// TwinCAT 3 PLC project Main
// ProgramVersion: 3.1.4023.0
// libraries:
//   Tc2_Standard, * (Beckhoff Automation GmbH)
//   Tc2_System, * (Beckhoff Automation GmbH)
//   Tc3_Module, * (Beckhoff Automation GmbH)
// project tree:
//   DUTs/ Controller.TcDUT, ControllerCmd.TcDUT, E_TriggerModes.TcDUT, E_PlayerID.TcDUT, E_ConnectionType.TcDUT, E_LedOptions.TcDUT, E_PulseOptions.TcDUT, E_Brightness.TcDUT, Point.TcDUT
//   GVLs/ Global.TcGVL
//   / PlcTask.TcTTO
//   POUs/ MAIN.TcPOU
// real-time tasks:
//   TASK PlcTask: cycle T#10ms, priority 20, ADS port 350

CONFIGURATION Main
    RESOURCE PLC ON TwinCAT3
        TASK PlcTask(INTERVAL := T#10ms, PRIORITY := 20);
        PROGRAM MAIN WITH PlcTask : MAIN;
    END_RESOURCE
END_CONFIGURATION

// ---- DUTs/Controller.TcDUT
TYPE Controller :
STRUCT
	LeftJoystickX : INT;
	LeftJoystickY : INT;
	RightJoystickX : INT;
	RightJoystickY : INT;
	LeftTrigger : INT;
	RightTrigger : INT;
	LeftBumper : BOOL;
	RightBumper : BOOL;
	ButtonTriangle : BOOL;
	ButtonCircle : BOOL;
	ButtonSquare : BOOL;
	ButtonCross : BOOL;
	LeftThumb : BOOL;
	RightThumb : BOOL;
	Share : BOOL;
	Options : BOOL;
	Ps : BOOL;
	DPadUp : BOOL;
	DPadDown : BOOL;
	DPadLeft : BOOL;
	DPadRight : BOOL;
	TouchBtn : BOOL;
	TrackPadTouch0Active : BOOL;
	TrackPadTouch1Active : BOOL;
	TrackPadTouch0ID : INT;
	TrackPadTouch1ID : INT;
	TrackPadTouch0X : INT;
	TrackPadTouch0Y : INT;
	TrackPadTouch1X : INT;
	TrackPadTouch1Y : INT;
	GyroPitch : INT;
	GyroYaw : INT;
	GyroRoll : INT;
	AccX : INT;
	AccY : INT;
	AccZ : INT;
	MicBtn : BOOL;
END_STRUCT
END_TYPE

// ---- DUTs/ControllerCmd.TcDUT
TYPE ControllerCmd :
STRUCT
	
	LedRed : INT := 255;
	LedGreen : INT;
	LedBlue : INT;
	Player : E_PlayerID;
	LedOptions : E_LedOptions;
	PulseOptions : E_PulseOptions;
	Brightness : E_Brightness;
	LeftHaptic : INT;
	RightHaptic : INT;
	LeftTriggerMode : E_TriggerModes;
	LeftTriggerLevel1 : INT;
	LeftTriggerLevel2 : INT;
	LeftTriggerLevel3 : INT;
	LeftTriggerLevel4 : INT;
	LeftTriggerLevel5 : INT;
	LeftTriggerLevel6 : INT;
	LeftTriggerLevel7 : INT;
	RightTriggerMode : E_TriggerModes;
	RightTriggerLevel1 : INT;
	RightTriggerLevel2 : INT;
	RightTriggerLevel3 : INT;
	RightTriggerLevel4 : INT;
	RightTriggerLevel5 : INT;
	RightTriggerLevel6 : INT;
	RightTriggerLevel7 : INT;
	MicLed : BOOL;
	MicMute : BOOL;
	
END_STRUCT
END_TYPE

// ---- DUTs/E_TriggerModes.TcDUT
{attribute 'qualified_only'}
TYPE E_TriggerModes :
(
	Off := 16#0, // no resistance
    Rigid := 16#1, // continous resistance
    Pulse := 16#2, // section resistance
    Rigid_A := 16#1 OR 16#20,
    Rigid_B := 16#1 OR 16#04,
    Rigid_AB := 16#1 OR 16#20 OR 16#04,
    Pulse_A := 16#2 OR 16#20,
    Pulse_B := 16#2 OR 16#04,
    Pulse_AB := 16#2 OR 16#20 OR 16#04,
    Calibration:= 16#FC
) INT;
END_TYPE

// ---- DUTs/E_PlayerID.TcDUT
{attribute 'qualified_only'}
TYPE E_PlayerID :
(
	player1 := 4,
    player2 := 10,
    player3 := 21,
    player4 := 27,
    all := 31
) INT;
END_TYPE

// ---- DUTs/E_ConnectionType.TcDUT
{attribute 'qualified_only'}
TYPE E_ConnectionType :
(
	BT := 16#00,
	USB := 16#01
) INT;
END_TYPE

// ---- DUTs/E_LedOptions.TcDUT
{attribute 'qualified_only'}
TYPE E_LedOptions :
(
	Off :=16#00,
    PlayerLedBrightness :=16#01,
    UninterrumpableLed :=16#02,
    Both := 16#01 OR 16#02
) INT;
END_TYPE

// ---- DUTs/E_PulseOptions.TcDUT
{attribute 'qualified_only'}
TYPE E_PulseOptions :
(
	Off :=16#00,
    FadeBlue :=16#01,
    FadeOut :=16#02
) INT;
END_TYPE

// ---- DUTs/E_Brightness.TcDUT
{attribute 'qualified_only'}
TYPE E_Brightness :
(
	high :=16#00,
    medium :=16#01,
    low :=16#02
) INT;
END_TYPE

// ---- DUTs/Point.TcDUT
TYPE Point :
STRUCT
	x : INT;
	y : INT;
END_STRUCT
END_TYPE

// ---- GVLs/Global.TcGVL
{attribute 'qualified_only'}
VAR_GLOBAL
	controller : Controller;
	controllerCmd : ControllerCmd;
	touchData : ARRAY [0..1,0..0] OF Point := [(x:=0,y:=0),(x:=0,y:=0)];
END_VAR

// ---- POUs/MAIN.TcPOU
PROGRAM MAIN
VAR
END_VAR

Global.touchData[0,0].x := Global.controller.TrackPadTouch0X;
Global.touchData[0,0].y := Global.controller.TrackPadTouch0Y;
Global.touchData[1,0].x := Global.controller.TrackPadTouch1X;
Global.touchData[1,0].y := Global.controller.TrackPadTouch1Y;

END_PROGRAM
